{attribute addProperty BoxType "EL7041-0001-0016"}
{attribute addProperty Id "ControlAT %Q*Control_D763B957445.5"}
{attribute addProperty CRC "782071841"}
{attribute addProperty SizeInBites "44"}
{attribute addProperty SizeInBytes "5.5"}
TYPE STM_Control_2E9D7821 :
STRUCT
	{attribute addProperty Name "Control"}
	Control AT %Q* : Control_D763B957;
END_STRUCT
END_TYPE

(* stored: Version 1.2.0.0, ProductVersion 3.1.4024.9
   DUT STM_Control_2E9D7821: Id {fafcf396-cda2-4703-9911-78f67b5a0b1a} *)
